(* CODESYS project GersSciPal_Project.project
   Company: io systems
   Title: GersSciPal_Project
   Description: application suivi de production
   Author: jl
   Version: 0.0.0.0

Project tree, tasks and I/O mapping:
  HMISCUxA5 : HMISCUxA5, Schneider Electric, order no. HMISCUxA5, version 3.5.3.59
      settings: OpcUa Enable = False
    application Application
      libraries: SysTimeRtc, 3.5.1.0 (System); ModbusTCP Slave, 3.5.3.50 (3S - Smart Software Solutions GmbH); 3S Storage, 3.5.3.0 (3S - Smart Software Solutions GmbH); BASIC, 3.3.4.0 (OSCAT)
      task MAST (cyclic, interval 20 ms, priority 15, watchdog 100 ms x 1) calls Prog_Main
      program Prog_Main [LD]
      Symbols
      999 - simulations/
        program random [LD]
        function block simulCounter [ST]
      200 - events & fifo/
        function block FB_fifoPushEvent [ST]
        program fifoManager [ST]
        function block eventManager [ST]
        function FC_fifoPush [ST]
      900 - utils/
        function CheckBounds [ST]
        function block TP_GSP [ST]
        function block Etat_Voyants [ST]
        function block counterWatch [ST]
        program CommunicationLife [ST]
      000 - data/
        global variables GVL
        data type _structModbusIn
        data type _structMessage
        data type alarmes
        data type _structVoyant
        data type _structModbusOut
        data type _structModbus
        data type _structIHMOFManager
        data type _structModbusMessage
      100 - time & com/
        program Modbus [LD]
        program timestamps [LD]
      300 - production/
        function block fabricationOrderManagement [ST]
    HMI Application
    Fonctions intégrées
      ES : ES, Schneider Electric, order no. IO, version 3.5.3.59
          input  iwES_Entr_e : WORD  // In
          output qwES_Sortie : WORD  // Out
      HSC : HSC, Schneider Electric, order no. HSC, version 3.5.3.59
      PTO_PWM : PTO_PWM, Schneider Electric, order no. PTO_PWM, version 3.5.3.59
    COM1
      SoMachine_Network_Manager : SoMachine-Network Manager, Schneider Electric, version 4.0.0.2
    Ethernet
      SoMachine_Network_Manager1 : SoMachine-Network Manager, Schneider Electric, version 4.0.0.2
    USB
      SoMachine_Network_Manager2 : SoMachine-Network Manager, Schneider Electric, version 4.0.0.2
    CAN
  Vijeo Designer Project Container Data
  Vijeo Designer Project Container
*)

// HMISCUxA5/Application/000 - data/_structModbusIn
TYPE _structModbusIn :
STRUCT
	ID: UDINT; // IDENTIFIANT DU MESSAGE AUTOMATE   0 à 3
    STATUT: INT; // ETAT A PRENDRE EN COMPTE         4 à 5
    lifeWD: INT; // MOT DE VIE  6 à 7
	rate: INT; // CADENCE THEORIQUE DE LA LIGNE
	reserve: INT;
END_STRUCT
END_TYPE

// HMISCUxA5/Application/000 - data/_structMessage
TYPE _structMessage :
STRUCT
	ihmOperations: STRING[8];
	ihmAlea: STRING[8];
	ihmLabels: STRING[32];

END_STRUCT
END_TYPE

// HMISCUxA5/Application/000 - data/alarmes
TYPE alarmes :
STRUCT
	attenteServeur: BOOL;
	attenteMariadb: BOOL;
	blocageMachine: BOOL;
	blocEvent: BOOL;
	blocOF: BOOL;
	nodeREDLife: BOOL;
END_STRUCT
END_TYPE

// HMISCUxA5/Application/000 - data/_structVoyant
TYPE _structVoyant :
STRUCT
	input: BOOL;
	change: BOOL;
	valeur: int;
END_STRUCT
END_TYPE

// HMISCUxA5/Application/000 - data/_structModbusOut
TYPE _structModbusOut :
STRUCT
	// VALEURS DES COMPTEURS
	CNT1: UDINT; // NOMBRE DE PIECES PRODUITES // de l'octet 8 à 11
	CNT2: UDINT; // NOMBRE DE PIECES PRODUITES MAIS PAS BONNES // de l'octet 12 à 15      
	
	// CONTENU DU MESSAGE
	MESSAGE: _structModbusMessage;
	
	// CADENCES ET SURVEILLANCES
	RUN: INT; // 2 octets - 74 à 75
	CRTHORODATAGE : UDINT; // 4 octets - 76 à 79
	CADENCE: UDINT;  // UNITE PAR HEURE --> CHRONO ENTRE DEUX PALETTE, TOUTES LES 2 MINUTES ON ENREGISTRE LA VALEUR DE CNT1 ; 4 octets - 80 à 83
	CADENCE_MOYENNE: UDINT; // UNITE PAR HEURE --> DIFFERENCE EN CNT1 ACTUEL - CNT1 D'IL Y A UNE HEURE ; 4 octets - 84 à 87 
	life: INT; // MOT DE VIE ; 2 octets - 88 à 89

END_STRUCT
END_TYPE

// HMISCUxA5/Application/000 - data/_structModbus
TYPE _structModbus :
STRUCT
	modbusIn: _structModbusIn;
	modbusOut: _structModbusOut;
END_STRUCT
END_TYPE

// HMISCUxA5/Application/000 - data/_structIHMOFManager
TYPE _structIHMOFManager :
	STRUCT
		startOF: BOOL; // commande démarrer OF
		stopOF: BOOL; // commande arrêter OF
		X0: BOOL; // attente lancement OF
		X1: BOOL; // lancement OF
		X2: BOOL; // OF en cours, attente arrêt OF
		X3: BOOL; // arrêt OF
		newOFEmpty: BOOL;
		seq: INT; // image du sequenceur
		newOF: STRING[12]; // nouvel OF à lancer
		cnt2: INT; // nombre de pièces défectueuses, saisi à l'arrêt de l'OF
	END_STRUCT
END_TYPE

// HMISCUxA5/Application/000 - data/_structModbusMessage
TYPE _structModbusMessage :
STRUCT
	ID: UDINT := 0; // 4 octets - 16 à 19
    STATUT: INT := 0; // 2 octets - 20 à 21
    OFNR: STRING[12] := '            '; // 13 octets - 22 à 33
    CODEM: STRING[8] := '        '; // 9 octets - 34 à 42
    OPERATION: STRING[8] := '        '; // 9 octets - 43 à 51
    ALEA: STRING[8] := '        '; // 9 octets - 52 à 60
    LIBELLE: STRING[32] := '                                '; // 17 octets - 52 à 67
	HORODATAGE: UDINT := 0; // 4 octets - 68 à 71 
	VALEUR: INT := 0; // 2 octets - 72 à 73
END_STRUCT
END_TYPE

// HMISCUxA5/Application/000 - data/GVL
VAR_GLOBAL
	Unixtime: UDINT; // Nombre de secondes depuis le 1er janvier 1970, lu sur l’horloge RTC de l’automate
	plcCycleTime: TIME;
	
	// table d'échange modbus avec Node-RED
	modbusInOut: _structModbus;
	startModbus: BOOL := TRUE;
	modbusError: BOOL := false;
	
	// données des messages et contenu de la FIFO
    fifoCount: INT := 0; // LONGUEUR REELLE DE LA PILE FIFO
	emptyMessage: _structModbusMessage; // CE MESSAGE DOIT TOUJOURS RESTER VIDE
	fifo: ARRAY[0..31] OF _structModbusMessage;
	
	// numéro d'OF de l'application
	OFNR: STRING[12] := '            ';
	
	// messages d'alarmes
	alm: alarmes;
	RPIOK: BOOL;
	DBOK: BOOL;
	NODEREDOK: BOOL;
	
	//Valeur Bouton IHM
	initFifoCount: BOOL;
	runAuto: BOOL;
	ihmButtons: ARRAY[0..15] OF BOOL;
	ihmOFManager: _structIHMOFManager;
	ihmOFRunning : BOOL;
	
	// gestion popup statut message
	closePopup: BOOL;
	
	// données gestion des voyants
	etatsVoyants: ARRAY[0..15] OF _structVoyant;
	
	// blocage machine
	AutorisationAuto AT %QX0.2 : BOOL;
	
END_VAR

VAR_GLOBAL CONSTANT
	fifoIndexMin: INT := 0;
    fifoIndexMax: INT := 31;
END_VAR

VAR_GLOBAL RETAIN PERSISTENT
	bypassAutoOut: BOOL;
	CNT1: UDINT;	// COMPTEUR DES PIECES CONFORMES
	CNT2: UDINT;	// COMPTEUR DES PIECES NON CONFORMES
	messageID: UDINT; // COMPTEUR DE MESSAGES
	CODEM: STRING[8];
	
	// PARAMETRES DE L'APPLICATION
	gvl_counterWatch_ptLife: TIME := T#20s;
	gvl_counterWatch_ptRate: TIME := T#2M;
	gvl_counterWatch_ptPercent: INT := 15;
	Param_minTime	: TIME := T#350MS;
	Param_maxTime	: TIME := T#750MS;
	Param_onOffTime	: TIME := T#2S;
	
	// RECETTE
	ihmMessages: ARRAY[0..31] OF _structMessage;
	
	// TITRES DES BOUTONS IHM
	buttons_FR: ARRAY[0..15] OF STRING[16];
	buttons_HU: ARRAY[0..15] OF STRING[16];
	buttons_EN: ARRAY[0..15] OF STRING[16];
	
END_VAR

// HMISCUxA5/Application/Prog_Main
PROGRAM Prog_Main
VAR
	
	em: eventManager;
	cw: counterWatch;
	fom: fabricationOrderManagement;
	
END_VAR

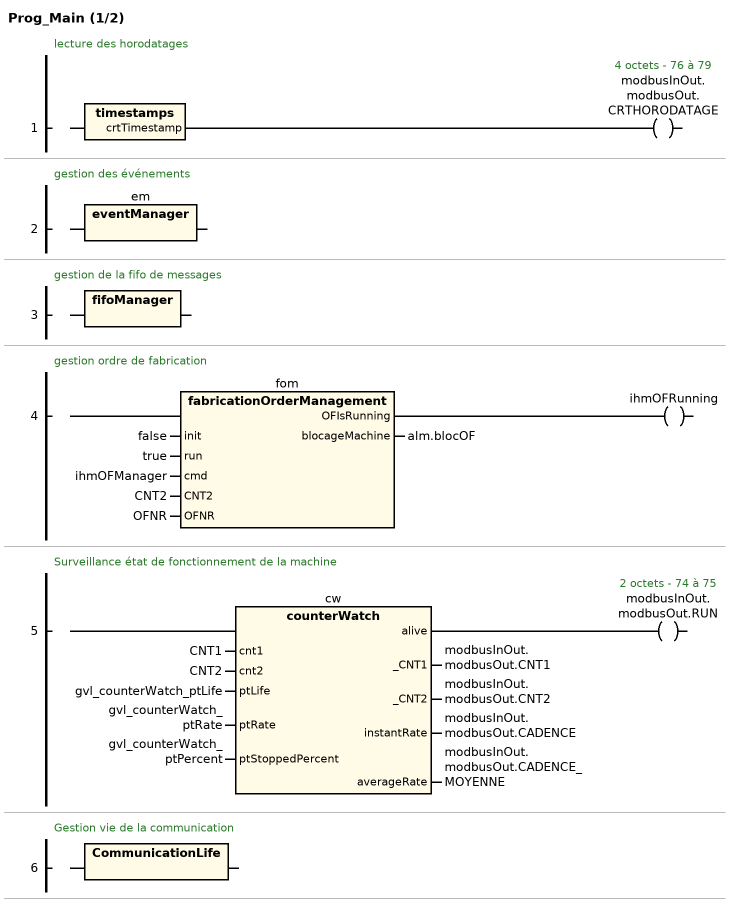
// NETWORK 1
// lecture des horodatages
//   modbusInOut.modbusOut.CRTHORODATAGE: 4 octets - 76 à 79
timestamps();
modbusInOut.modbusOut.CRTHORODATAGE := timestamps.crtTimestamp;

// NETWORK 2
// gestion des événements
em(); // eventManager

// NETWORK 3
// gestion de la fifo de messages
fifoManager();

// NETWORK 4
// gestion ordre de fabrication
//   CNT2: COMPTEUR DES PIECES NON CONFORMES
//   OFNR: numéro d'OF de l'application
fom(
    init := false,
    run := true,
    cmd := ihmOFManager,
    CNT2 := CNT2,
    OFNR := OFNR,
    blocageMachine => alm.blocOF); // fabricationOrderManagement
ihmOFRunning := fom.OFIsRunning;

// NETWORK 5
// Surveillance état de fonctionnement de la machine
//   CNT1: COMPTEUR DES PIECES CONFORMES
//   CNT2: COMPTEUR DES PIECES NON CONFORMES
//   gvl_counterWatch_ptLife: PARAMETRES DE L'APPLICATION
//   modbusInOut.modbusOut.CNT1: NOMBRE DE PIECES PRODUITES // de l'octet 8 à 11
//   modbusInOut.modbusOut.CNT2: NOMBRE DE PIECES PRODUITES MAIS PAS BONNES // de l'octet 12 à 15
//   modbusInOut.modbusOut.CADENCE: UNITE PAR HEURE --> CHRONO ENTRE DEUX PALETTE, TOUTES LES 2 MINUTES ON ENREGISTRE LA VALEUR DE CNT1 ; 4 octets - 80 à 83
//   modbusInOut.modbusOut.CADENCE_MOYENNE: UNITE PAR HEURE --> DIFFERENCE EN CNT1 ACTUEL - CNT1 D'IL Y A UNE HEURE ; 4 octets - 84 à 87
//   modbusInOut.modbusOut.RUN: 2 octets - 74 à 75
cw(
    cnt1 := CNT1,
    cnt2 := CNT2,
    ptLife := gvl_counterWatch_ptLife,
    ptRate := gvl_counterWatch_ptRate,
    ptStoppedPercent := gvl_counterWatch_ptPercent,
    _CNT1 => modbusInOut.modbusOut.CNT1,
    _CNT2 => modbusInOut.modbusOut.CNT2,
    instantRate => modbusInOut.modbusOut.CADENCE,
    averageRate => modbusInOut.modbusOut.CADENCE_MOYENNE); // counterWatch
modbusInOut.modbusOut.RUN := cw.alive;

// NETWORK 6
// Gestion vie de la communication
CommunicationLife();

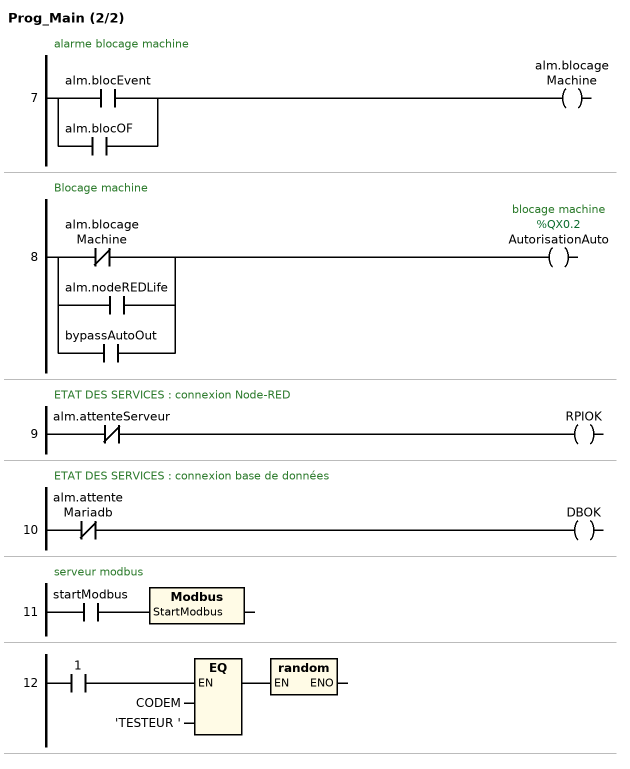
// NETWORK 7
// alarme blocage machine
alm.blocageMachine := alm.blocEvent OR alm.blocOF;

// NETWORK 8
// Blocage machine
//   AutorisationAuto: blocage machine | AT %QX0.2
AutorisationAuto := NOT alm.blocageMachine OR alm.nodeREDLife OR bypassAutoOut;

// NETWORK 9
// ETAT DES SERVICES : connexion Node-RED
RPIOK := NOT alm.attenteServeur;

// NETWORK 10
// ETAT DES SERVICES : connexion base de données
DBOK := NOT alm.attenteMariadb;

// NETWORK 11
// serveur modbus
Modbus(StartModbus := startModbus);

// NETWORK 12
IF 1 AND CODEM = 'TESTEUR ' THEN random(); END_IF

END_PROGRAM

// HMISCUxA5/Application/100 - time & com/timestamps
PROGRAM timestamps
VAR_OUTPUT
	crtTimestamp: UDINT;
END_VAR
VAR
	pResult :UDINT;
	tBool: BOOL;
	plcCyleTime: OSCAT_BASIC.CYCLE_TIME;
	ct_min: TIME;
	ct_max: TIME;
	systime: TIME;
	sysdays: INT;
	cycles:DWORD;
	tmpTime: DWORD;
END_VAR

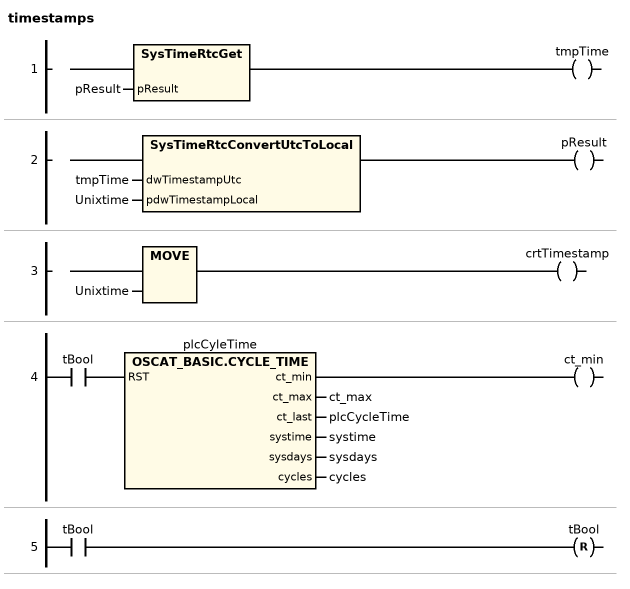
// NETWORK 1
tmpTime := SysTimeRtcGet(pResult := pResult);

// NETWORK 2
//   Unixtime: Nombre de secondes depuis le 1er janvier 1970, lu sur l’horloge RTC de l’automate
pResult := SysTimeRtcConvertUtcToLocal(dwTimestampUtc := tmpTime, pdwTimestampLocal := Unixtime);

// NETWORK 3
//   Unixtime: Nombre de secondes depuis le 1er janvier 1970, lu sur l’horloge RTC de l’automate
crtTimestamp := Unixtime;

// NETWORK 4
plcCyleTime(
    RST := tBool,
    ct_max => ct_max,
    ct_last => plcCycleTime,
    systime => systime,
    sysdays => sysdays,
    cycles => cycles); // OSCAT_BASIC.CYCLE_TIME
ct_min := plcCyleTime.ct_min;

// NETWORK 5
tBool R= tBool;

END_PROGRAM

// HMISCUxA5/Application/200 - events & fifo/eventManager
FUNCTION_BLOCK eventManager
VAR_INPUT
END_VAR
VAR_OUTPUT
END_VAR
VAR
	fifoPush: ARRAY[0..31] OF FB_fifoPushEvent;
	etatsVoyantsFB: ARRAY[0..15] OF Etat_Voyants;
	oldTmpBool: ARRAY[0..31] OF BOOL;
	tmpMessage: _structModbusMessage;
	tonResetButton11: Standard.TON;
	seqStop: INT := 0;
	msgIdStop: INT := 0;
END_VAR
VAR_TEMP
	tmpBool: BOOL;
	i: INT := 0;
	j: INT := 7;
END_VAR

tonResetButton11(in := ihmButtons[11], pt := T#500MS);
IF tonResetButton11.Q THEN
	ihmButtons[11] := FALSE;
END_IF

FOR i := 0 TO 31 BY +1 DO
	// SELECTION DE L'ENTREE AUTOMATE OU DU BOUTON IHM
	CASE i OF
		0: tmpBool:= %IX0.0;		
		1: tmpBool:= %IX0.1;		
		2: tmpBool:= %IX0.2;		
		3: tmpBool:= %IX0.3; 	
		4: tmpBool:= %IX0.4;		
		5: tmpBool:= %IX0.5;		
		6: tmpBool:= %IX0.6;		
		7: tmpBool:= %IX0.7;		
		8: tmpBool:= %IX1.0;
		9: tmpBool:= %IX1.1;
		10: tmpBool:= %IX1.2;
		11: tmpBool:= %IX1.3;
		12: tmpBool:= %IX1.4;
		13: tmpBool:= %IX1.5;
		14: tmpBool:= %IX1.6;
		15: tmpBool:= %IX1.7;
		16..31: tmpBool:= ihmButtons[i - 16];
	END_CASE
	
	// TRAITEMENT CAS PARTICULIER : OPERATION COMPTEUR
	IF ihmMessages[i].ihmOperations = 'COMPTEUR' THEN 
		
		// UNIQUEMENT ENTREE AUTOMATE
		IF i < 16 THEN
			// COMPTEUR DES PIECES CONFORMES
			IF ihmMessages[i].ihmAlea = 'CNT1    ' THEN
				IF tmpBool AND NOT oldTmpBool[i] THEN
					CNT1 := CNT1 + 1;
				END_IF;

			// COMPTEUR DES PIECES NON CONFORMES
			ELSIF ihmMessages[i].ihmAlea = 'CNT2    ' THEN
				IF tmpBool AND NOT oldTmpBool[i] THEN
					CNT2 := CNT2 + 1;
				END_IF;
			END_IF;
			
		END_IF;

	// TRAITEMENT CAS PARTICULIER : ENTREE AUTOMATE IMAGE D'UN VOYANT
	ELSIF ihmMessages[i].ihmOperations = 'VOYANT  ' THEN 
		
		// UNIQUEMENT ENTREE AUTOMATE
		IF i < 16 THEN
			// fonction de gestion de voyant
			etatsVoyantsFB[i](input := tmpBool, etatV := etatsVoyants[i]); 
		
			// DETECTION DERNIER CARACTERE DE LA CHAINE ALEA
			FOR j := 7 TO 0 BY -1 DO  
				IF ihmMessages[i].ihmAlea[j] <> 32 THEN
					EXIT;
				END_IF;
			END_FOR;
			// ECRITURE DE LA VALEUR DU VOYANT
			ihmMessages[i].ihmAlea[j] := BYTE#48 + INT_TO_BYTE(etatsVoyants[i].valeur); 
			
			// INSERTION DU MESSAGE DANS LA FIFO
			fifoPush[i](
				insert := etatsVoyants[i].change, 
				message:= ihmMessages[i]
			);
		END_IF;
		
	// TRAITEMENT CAS PARTICULIER : MESSAGES SYSTEME
	ELSIF ihmMessages[i].ihmOperations = 'RUN     ' THEN
		
		// MESSAGE 'RUNAUTO'
		IF ihmMessages[i].ihmAlea = 'RUNAUTO ' THEN
			tmpBool := modbusInOut.modbusOut.RUN > 0;
			fifoPush[i](
				insert := tmpBool,
				message:= ihmMessages[i]
			);
			
			// Blocage fonctionnement machine sur front descendant état de marche machine
			IF NOT tmpBool AND oldTmpBool[i] THEN
				seqStop := 1;
				// mémorisation horodatage arrêt machine
				tmpMessage.HORODATAGE := Unixtime;
				
			ELSIF tmpBool AND NOT oldTmpBool[i] AND seqStop = 1 THEN
				ihmButtons[11] := TRUE;
				
			END_IF; 
			
		END_IF;
		
	// CAS GENERAL : ENTREES AUTOMATE, NE DEBLOQUENT PAS LA MACHINE
	ELSIF i < 16 THEN
		// cas général
		fifoPush[i](
			insert := tmpBool,
			message:= ihmMessages[i]
		);
		
	// CAS GENERAL : BOUTONS IHM
	ELSE
		CASE seqStop OF
			0: // cas général
				fifoPush[i](
					insert := tmpBool,
					message:= ihmMessages[i]
				);
			
			1: // machine bloquée, attente sélection bouton ou redémarrage machine
				IF tmpBool AND NOT oldTmpBool[i] THEN
					msgIdStop := i;
					tmpMessage.OPERATION := ihmMessages[i].ihmOperations;
					tmpMessage.ALEA := ihmMessages[i].ihmAlea;
					tmpMessage.LIBELLE := ihmMessages[i].ihmLabels;
					// tmpMessage.horodatage a été saisi au front montant de alm.blocEvent, ligne 82
					tmpMessage.VALEUR := 1;
					FC_fifoPush(
						message := tmpMessage
					);
					seqStop := 2;
				END_IF
				
			2: // machine bloquée, attente remise à 0 du bouton IHM
				IF i = msgIdStop AND NOT tmpBool AND oldTmpBool[i] THEN
					tmpMessage.OPERATION := ihmMessages[i].ihmOperations;
					tmpMessage.ALEA := ihmMessages[i].ihmAlea;
					tmpMessage.LIBELLE := ihmMessages[i].ihmLabels;
					tmpMessage.horodatage := Unixtime;
					tmpMessage.VALEUR := 0;
					FC_fifoPush(
						message := tmpMessage
					);
					seqStop := 0;
				END_IF
				
			ELSE
				seqStop := 0;
			
		END_CASE
		
	END_IF;
	
	// MISE A JOUR DES ETATS PRECEDENTS
	oldTmpBool[i] := tmpBool;
	
END_FOR
alm.blocEvent := seqStop >= 1;

// REMPLACEMENT CARACTERE 0 PAR UN ESPACE DANS LE CODEM (VENANT DE LA RECETTE)
FOR i := 0 TO 7 BY +1 DO
	IF CODEM[ i ] = 0 THEN
		CODEM[ i ] := 32;
	END_IF
END_FOR;

END_FUNCTION_BLOCK

// HMISCUxA5/Application/200 - events & fifo/FC_fifoPush
FUNCTION FC_fifoPush : int
VAR_INPUT
	message: _structModbusMessage;
END_VAR

// NE DOIT ETRE APPELEE QUE SUR FRONT MONTANT OU DESCENDANT !!!

IF message.OPERATION = '        ' OR message.ALEA = '        ' OR message.LIBELLE = '                                ' THEN
	RETURN;
END_IF

// ENREGISTREMENT DU MESSAGE
fifo[ fifoCount ] := message;

// MISE A JOUR DES VALEURS PAR DEFAUT
fifo[ fifoCount ].ID := messageID;
fifo[ fifoCount ].STATUT := 2;
fifo[ fifoCount ].OFNR := OFNR;
fifo[ fifoCount ].CODEM := CODEM;

// MISE À JOUR DE LA LONGUEUR DE LA PILE
IF fifoCount < fifoIndexMax THEN
	fifoCount := fifoCount + 1;
END_IF;

// INCRÉMENT DU COMPTEUR DE MESSAGE
messageID := messageID + 1;
IF messageID > 32765 THEN
	messageID := 0;
END_IF;

FC_fifoPush := 0;

END_FUNCTION

// HMISCUxA5/Application/200 - events & fifo/FB_fifoPushEvent
FUNCTION_BLOCK FB_fifoPushEvent
VAR_INPUT
	insert: BOOL;
	message: _structMessage;
END_VAR
VAR
	memInsert: BOOL;
END_VAR
VAR_TEMP
	tmpMessage: _structModbusMessage;
END_VAR

// CONTROLE DU CONTENU DU MESSAGE
IF message.ihmOperations = '        ' OR message.ihmAlea = '        ' OR message.ihmLabels = '                                '
	OR CODEM = '        ' THEN
	RETURN;
END_IF

// INSERTION MESSAGE SUR CHANGEMENT D'ETAT DE L'ENTREE INSERT
IF insert AND NOT memInsert  OR NOT insert AND memInsert THEN
	// DÉFINITION DU MESSAGE
	tmpMessage.OPERATION := message.ihmOperations;
	tmpMessage.ALEA := message.ihmAlea;
	tmpMessage.LIBELLE := message.ihmLabels;
	tmpMessage.HORODATAGE := Unixtime;
	IF insert THEN
		tmpMessage.VALEUR := 1;
	ELSE
		tmpMessage.VALEUR := 0;
	END_IF;
	
	FC_fifoPush(
		message := tmpMessage
	);

END_IF;
memInsert := insert;

END_FUNCTION_BLOCK

// HMISCUxA5/Application/900 - utils/Etat_Voyants
FUNCTION_BLOCK Etat_Voyants
VAR_INPUT
	input: BOOL;
END_VAR
VAR_IN_OUT
	etatV: _structVoyant;
END_VAR
VAR
	old_input: BOOL;
	tmp: INT := 0;
	old_tmp: INT := 0;
	time_on: TIME;
	time_off: TIME;
	last_time_on: TIME;
	last_time_off: TIME;
	tonChange : Standard.TON;
	seq: INT;
	backup: INT;
END_VAR
VAR_TEMP
	minTime		: TIME;
	maxTime		: TIME;
	onOffTime	: TIME;
	cycleTime	: TIME;
	limitTime	: TIME;
END_VAR

minTime := Param_minTime;// T#250MS;
maxTime := Param_maxTime; // T#500MS;
onOffTime := Param_onOffTime; // T#2S;
cycleTime := onOffTime; // Param_cycleTime; // T#2S;
limitTime := T#30S;

etatV.input := input;

IF etatv.input AND NOT old_input THEN
	last_time_off := time_off;
	time_off := T#0S;
END_IF
IF NOT etatv.input AND old_input THEN
	last_time_on := time_on;
	time_on := T#0S;
END_IF

IF etatv.input THEN
	IF time_on < limitTime THEN
		time_on := time_on + plcCycleTime;
	END_IF;
ELSE
	IF time_off < limitTime THEN
		time_off := time_off + plcCycleTime;
	END_IF;
END_IF

IF time_on > onOffTime THEN
	tmp := 1;
	
ELSIF time_off > onOffTime THEN
	tmp := 0;
	
ELSIF last_time_on > minTime AND last_time_off > minTime THEN
	IF last_time_on > maxTime AND last_time_off > maxTime THEN
		tmp := 3;
	ELSE
		tmp := 2;
	END_IF;
END_IF; 

tonChange(in := etatV.valeur <> tmp, pt := cycleTime);
CASE seq OF
	0: 
		IF tonChange.Q THEN
			old_tmp := etatV.valeur;
			backup := tmp;
			seq := 1;
		END_IF
		
	1: 
		etatV.change := FALSE;
		seq := 2;
		
	2:
		etatV.valeur := backup;
		etatV.change := TRUE;
		seq := 0;
		
	ELSE
		seq := 0;
			 
END_CASE

old_input := etatv.input;

END_FUNCTION_BLOCK

// HMISCUxA5/Application/200 - events & fifo/fifoManager
PROGRAM fifoManager
VAR
	i: INT;
	TON_STEP2: Standard.TON;
	TON_STEP3: Standard.TON;
	TON_STEP4: Standard.TON;
	TON_STEP6: Standard.TON;
	TON_STEP80: Standard.TON;
	TON_STEP81: Standard.TON;
	cycleTime: TIME := T#500MS;
	timeoutNodeRED: TIME := T#5S;
	timeoutDB: TIME := T#5S;
	resumeTime: TIME := T#2S;
	errServerCnt: INT := 0;
	errMariadDBCnt: INT := 0;
	maxErr: INT := 5;
END_VAR

// RECHERCHE DE L’INDICE DU PREMIER CHAMP VIDE EN PARTANT DU BAS DE LA PILE
// EXECUTER CETTE FONCTION UNIQUEMENT APRES LA MISE EN RUN DE L'AUTOMATE OU A LA DEMANDE
// PAR UN BOUTON IHM SI FIFOCOUNT EST PERDU
IF initFifoCount THEN
	FOR i := fifoIndexMax TO fifoIndexMin BY -1 DO
    	IF fifo[ i ].STATUT > 0 THEN
        	fifoCount := i + 1;
    	END_IF;
	END_FOR;	
	initFifoCount := FALSE;
END_IF

// TEMPORISATION CONTROLE COMMUNICATION
TON_STEP2( IN := fifo[ fifoIndexMin ].STATUT = 2, PT := cycleTime);
TON_STEP3( IN := fifo[ fifoIndexMin ].STATUT = 3, PT := timeoutNodeRED);
TON_STEP4( IN := fifo[ fifoIndexMin ].STATUT = 4, PT := timeoutDB);
TON_STEP6( IN := fifo[ fifoIndexMin ].STATUT = 6, PT := cycleTime);
TON_STEP80( IN := fifo[ fifoIndexMin ].STATUT = 80, PT := resumeTime);
TON_STEP81( IN := fifo[ fifoIndexMin ].STATUT = 81, PT := resumeTime);

// GESTION ACTIVITE PREMIER MESSAGE DANS LA FIFO
CASE fifo[ fifoIndexMin ].STATUT OF
	0:	// STATUS 0 = PAS DE MESSAGE
		;
		
	1:	// STATUS 1 = MESSAGE EN COURS DE SAISIE 
		;
		
	2: 	// STATUS 2 = MESSAGE EN ATTENTE DE TRANSMISSION
		IF TON_STEP2.Q THEN
			// MISE À DISPOSITION DU PREMIER MESSAGE DE LA PILE POUR SRV-IOT
			fifo[ fifoIndexMin ].STATUT := 3;
		END_IF;
		
	3:	// STATUS 3 = ATTENTE PRISE EN COMPTE MESSAGE PAR NODE-RED
		// SRV-IOT A LU LE MESSAGE
		IF modbusInout.modbusIn.ID = fifo[ fifoIndexMin ].ID AND modbusInout.modbusIn.STATUT = 4 THEN
			errServerCnt := 0;
			fifo[ fifoIndexMin ].STATUT := 4;
			
		ELSIF TON_STEP3.Q THEN
			// TIME OUT : Node-RED n'a pas répondu assez rapidement : annulation et relance
			errServerCnt := errServerCnt + 1;
			fifo[fifoIndexMin].STATUT := 80;
			
		END_IF;
		
	4: // STATUS 4 = ATTENTE RETOUR ENREGISTREMENT DANS LA BASE DE DONNEES
		alm.attenteServeur := FALSE;
		// LE MESSAGE A ÉTÉ ENREGISTRÉ DANS LA BASE DE DONNÉES
		IF modbusInout.modbusIn.ID = fifo[ fifoIndexMin ].ID AND modbusInout.modbusIn.STATUT = 5 THEN
			errMariadDBCnt := 0;
			fifo[ fifoIndexMin ].STATUT := 5;
			
		ELSIF TON_STEP4.Q THEN
			// TIME OUT : Node-RED n'a pas répondu dans les temps : annulation et relance
			errMariadDBCnt := errMariadDBCnt + 1;
			fifo[ fifoIndexMin ].STATUT := 81;
			
		END_IF;
		
	5:	// STATUS 5 = ARCHIVAGE MESSAGE ET ON PASSE AU SUIVANT
		alm.attenteMariadb := FALSE;
		// DECALAGE DE LA FIFO DE MESSAGES, ECRASEMENT DU MESSAGE EN COURS DE TRAITEMENT...
		FOR i := fifoIndexMin TO fifoIndexMax - 1 BY 1 DO
			fifo[ i ] := fifo[ i + 1];
		END_FOR;
		fifo[ fifoIndexMax ] := emptyMessage;
		
		// MISE À JOUR DE LA LONGUEUR RÉELLE DE LA PILE
		IF fifoCount > fifoIndexMin THEN
			fifoCount := fifoCount - 1;
		END_IF;
		
		// fermeture popup statut message
		closePopup := not closePopup;

	80:	// STATUT 80 : TIME OUT PRISE EN COMPTE DU MESSAGE PAR NODE RED
		alm.attenteServeur := TRUE;
		IF TON_STEP80.Q THEN
			fifo[ fifoIndexMin ].STATUT := 2;
		ELSIF errServerCnt >= maxErr THEN
			errServerCnt := 0;
			fifo[ fifoIndexMin ].STATUT := 5;
		END_IF;
		
	81: // STATUT 81 : TIME OUT ENREGISTREMENT MESSAGE DANS LA BASE DE DONNEES
		alm.attenteMariadb := TRUE;
		IF TON_STEP81.Q THEN
			fifo[ fifoIndexMin ].STATUT := 2;
		ELSIF errMariadDBCnt >= maxErr THEN
			errMariadDBCnt := 0;
			fifo[ fifoIndexMin ].STATUT := 5;
		END_IF;
		
	ELSE
		fifo[ fifoIndexMin ].STATUT := 0;
		
END_CASE;

// transmission message en modbus
modbusInOut.modbusOut.MESSAGE.STATUT := fifo[ fifoIndexMin ].STATUT;
IF fifo[ fifoIndexMin ].STATUT <= 0 THEN
	modbusInOut.modbusOut.MESSAGE.CODEM := CODEM;
	modbusInOut.modbusOut.MESSAGE.OFNR := OFNR;
	modbusInOut.modbusOut.MESSAGE.HORODATAGE := Unixtime;
ELSE
	modbusInOut.modbusOut.MESSAGE.ID :=  fifo[ fifoIndexMin ].ID;
	modbusInOut.modbusOut.MESSAGE.CODEM :=  fifo[ fifoIndexMin ].CODEM;
	modbusInOut.modbusOut.MESSAGE.OFNR :=  fifo[ fifoIndexMin ].OFNR;
	modbusInOut.modbusOut.MESSAGE.HORODATAGE :=  fifo[ fifoIndexMin ].HORODATAGE;
	modbusInOut.modbusOut.MESSAGE.OPERATION :=  fifo[ fifoIndexMin ].OPERATION;
	modbusInOut.modbusOut.MESSAGE.ALEA :=  fifo[ fifoIndexMin ].ALEA;
	modbusInOut.modbusOut.MESSAGE.LIBELLE :=  fifo[ fifoIndexMin ].LIBELLE;
	modbusInOut.modbusOut.MESSAGE.VALEUR :=  fifo[ fifoIndexMin ].VALEUR;
END_IF;

END_PROGRAM

// HMISCUxA5/Application/100 - time & com/Modbus
PROGRAM Modbus
VAR_IN_OUT
	StartModbus: BOOL;
END_VAR
VAR
	reset: BOOL;
	xBusy: BOOL;
	modbusInADR: POINTER TO WORD := ADR(modbusInOut);
	modbusRegistersADR: POINTER TO WORD:= ADR(modbusInOut.modbusIn.ID);
	ByClientConnection: BYTE;
	uiInputDataSize: UINT := 8; // A ADAPTER
	uiOutputDataSize: UINT := 108; // A ADAPTER
	TON_Start: TON;
	TON_Start_ET: TIME;
	ModbusServer_1 : ModbusServer;

END_VAR

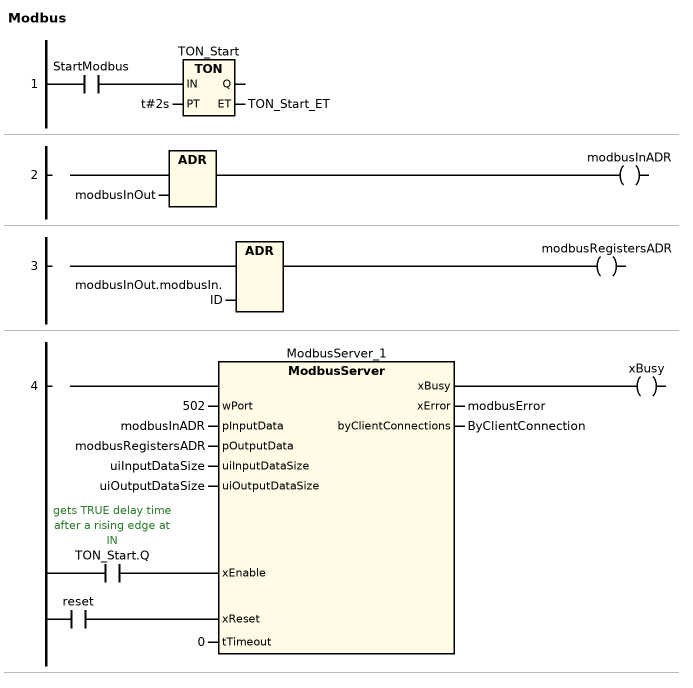
// NETWORK 1
TON_Start(IN := StartModbus, PT := t#2s, ET => TON_Start_ET); // TON

// NETWORK 2
//   modbusInOut: table d'échange modbus avec Node-RED
modbusInADR := ADR(modbusInOut);

// NETWORK 3
//   modbusInOut.modbusIn.ID: IDENTIFIANT DU MESSAGE AUTOMATE 0 à 3
modbusRegistersADR := ADR(modbusInOut.modbusIn.ID);

// NETWORK 4
//   uiInputDataSize: A ADAPTER
//   uiOutputDataSize: A ADAPTER
//   TON_Start.Q: gets TRUE delay time after a rising edge at IN
ModbusServer_1(
    wPort := 502,
    pInputData := modbusInADR,
    pOutputData := modbusRegistersADR,
    uiInputDataSize := uiInputDataSize,
    uiOutputDataSize := uiOutputDataSize,
    xEnable := TON_Start.Q,
    xReset := reset,
    tTimeout := 0,
    xError => modbusError,
    byClientConnections => ByClientConnection); // ModbusServer
xBusy := ModbusServer_1.xBusy;

END_PROGRAM

// HMISCUxA5/Application/300 - production/fabricationOrderManagement
FUNCTION_BLOCK fabricationOrderManagement
VAR_INPUT
	init: BOOL;
	run: BOOL;
END_VAR
VAR_OUTPUT
	OFIsRunning: BOOL;
	blocageMachine: BOOL;
END_VAR
VAR_IN_OUT
	cmd: _structIHMOFManager;
	CNT2: UDINT;
	OFNR: STRING[12];
END_VAR
VAR
	seq: INT;
END_VAR

// initialisations
OFIsRunning := FALSE;
blocageMachine := TRUE;

IF init THEN
	seq := 0;
	RETURN;
END_IF

// désactivation des transitions
IF NOT run THEN
	JMP end;
END_IF

// sequence
CASE seq OF
	0: // attente lancement OF
		IF cmd.newOF <> '            ' AND cmd.startOF THEN
			seq := 10;
		
		// si OF enregistré au démarrage, on l'arrête
		ELSIF OFNR <> '            ' THEN
			seq := 30;
			
		END_IF;
		
	10: // enregistrement du nouvel OF
		OFNR := cmd.newOF;
		cmd.startOF := FALSE;
		cmd.stopOF := FALSE;
		cmd.newOF := '            ';
		cmd.cnt2 := 0;
		seq := 20;
		
	20: // OF en cours
		OFIsRunning := TRUE;
		blocageMachine := FALSE;
		IF cmd.stopOF THEN
			seq := 30;
		END_IF;
		
	30: // arrêt OF en cours
		OFNR := '            ';
		cmd.startOF := FALSE;
		cmd.stopOF := FALSE;
		cmd.newOF := '            ';
		CNT2 := CNT2 + INT_TO_UDINT(cmd.cnt2);
		cmd.cnt2 := 0;
		seq := 0;
		
	ELSE
		seq := 0;
END_CASE

// mise à jour des recopies
end:
cmd.seq := seq / 10;
cmd.X0 := seq = 0;
cmd.X1 := seq = 10;
cmd.X2 := seq = 20;
cmd.X3 := seq = 30;
cmd.newOFEmpty := cmd.newOF = '            ';

END_FUNCTION_BLOCK

// HMISCUxA5/Application/900 - utils/counterWatch
FUNCTION_BLOCK counterWatch
VAR_INPUT
	cnt1: UDINT;
	cnt2: UDINT;
	ptLife: TIME;
	ptRate: TIME;
	ptStoppedPercent: INT;
END_VAR
VAR_OUTPUT
	alive: INT;
	_CNT1: UDINT;
	_CNT2: UDINT;
	instantRate: UDINT;
	averageRate: UDINT;
END_VAR
VAR
	TP_Life: TP_GSP;
	tonRate: TON;
	_ptLife: TIME;
	_ptRate: TIME;
	seq : INT;
	i : INT;
	tmpIndex: INT;
	oldCnt: UDINT;
	counts: ARRAY[0..59] OF UDINT;
	tmpReal: REAL;
END_VAR

// recopie des compteurs en sortie
_cnt1 := cnt1;
_cnt2 := cnt2;

// calcul du temps entre deux unités de cadences
_ptLife := ptLife;
IF modbusInOut.modbusIn.rate > 0 AND ptStoppedPercent > 0 AND  ptStoppedPercent < 100 THEN
	tmpReal := 3600.0 / (INT_TO_REAL(modbusInOut.modbusIn.rate) * (INT_TO_REAL(ptStoppedPercent) / 100.0)) * 1000.0; // Temps entre deux unités en millisecondes, temps mini = ptStoppedPercent de la cadence totale
	IF tmpReal > 0 THEN
		_ptLife := REAL_TO_TIME(tmpReal);
	END_IF
END_IF

// contrôle de la vie du compteur
TP_Life(in := cnt1 <> oldCnt, pt := _ptLife);
IF TP_Life.Q THEN
	alive := 1;
ELSE
	alive := 0;
END_IF
oldCnt := cnt1;

// init tableau en cas de remise à 0 du compteur
IF cnt1 < counts[0] THEN
	FOR i := 0 TO 29 BY 1 DO
		counts[i] := 0;
	END_FOR
END_IF

IF ptRate <= T#0S THEN
	return;
END_IF
_ptRate := ptRate;
IF _ptRate < T#1M THEN
	_ptRate := T#1M;
END_IF
IF _ptRate > T#1H THEN
	_ptRate := T#1H;
END_IF

// temps entre deux mesures de la cadence
tonRate(in := seq = 0, pt := _ptRate);

// séquence mesures de la cadence
CASE seq OF
	0:	// ATTENTE TEMPO CADENCE
		IF tonRate.Q THEN
			seq := 10;
		END_IF
		
	10: // INTEGRATION DE LA DERNIERE VALEUR DU COMPTEUR
		FOR i := 59 TO 1 BY -1 DO
			counts[i] := counts[i - 1];
		END_FOR
		counts[0] := cnt1;
		
		// CALCUL CADENCE INSTANTANEE
		// interdiction division par 0 et valeur négative
		IF _ptRate > T#0S AND counts[0] >= counts[1] THEN
			instantRate := (counts[0] - counts[1]) * TIME_TO_UDINT(T#1H) / TIME_TO_UDINT(_ptRate);
		ELSE
			instantRate := 0;
		END_IF
		
		// CALCUL DE LA CADENCE A L'HEURE
		// interdiction division par 0
		IF _ptRate > T#0S THEN
			tmpIndex := UDINT_TO_INT(TIME_TO_UDINT(T#1H) / TIME_TO_UDINT(_ptRate)) - 1;
			
			// tmpIndex doit être dans les limites du tableau
			IF tmpIndex > 0 AND tmpIndex <= 59 THEN
				
				// interdiction valeur négative
				IF counts[0] >= counts[tmpindex] THEN
					averageRate := (counts[0] - counts[tmpIndex]);
				ELSE
					averageRate := 0;
				END_IF
			ELSE
				averageRate := 0;
			END_IF;
		ELSE
			averageRate := 0;
		END_IF
		seq := 0;
		
	ELSE
		seq := 0;
END_CASE

END_FUNCTION_BLOCK

// HMISCUxA5/Application/900 - utils/TP_GSP
FUNCTION_BLOCK TP_GSP
VAR_INPUT
	IN: BOOL;
	PT: TIME;
END_VAR
VAR_OUTPUT
	Q: BOOL;
	ET: TIME;
END_VAR
VAR
	aux_in: BOOL;
	seq: INT;
	lastStart: TIME;
END_VAR

IF in AND NOT aux_in THEN
	lastStart := UDINT_TO_TIME(unixtime) * 1000;
	et := T#0s;
END_IF 
aux_in := in;

Q := FALSE;
CASE seq OF
	0:
		IF in THEN
			seq := 1;
		END_IF
		
	1:
		q := TRUE; 
		IF ET < PT THEN
			ET := UDINT_TO_TIME(unixtime) * 1000 - laststart;
		ELSE
			seq := 2;
		END_IF
		
	2:
		IF NOT in THEN
			seq := 0;
		END_IF
		
END_CASE

END_FUNCTION_BLOCK

// HMISCUxA5/Application/900 - utils/CommunicationLife
PROGRAM CommunicationLife
VAR
	oldReceivedLife: INT;
	seq: INT := 0;
	filterTime: TIME;
	TONLife: Standard.TON;
	TOFLife: Standard.TOF;
	ton_1: TON;
	ton_2: TON;
END_VAR

// création de la vie
IF modbusInOut.modbusOut.life < 999 THEN
	modbusInOut.modbusOut.life := modbusInOut.modbusOut.life + 1;
ELSE
	modbusInOut.modbusOut.life := 0;
END_IF

// surveillance vie Node-RED
filterTime := T#2S;
TONLife(in := modbusInOut.modbusIn.lifeWD = oldReceivedLife, pt := filterTime);
TOFLife(in := TONLife.Q, pt := filterTime);
oldReceivedLife := modbusInOut.modbusIn.lifeWD;

alm.nodeREDLife := FALSE; // TOFLife.Q;
NODEREDOK := NOT alm.nodeREDLife;

IF NODEREDOK THEN
	seq := 0;
	StartModbus := not modbusError;
	RETURN;
END_IF

ton_1(in := seq = 0 AND alm.nodeREDLife, pt := T#60S);
ton_2(in := seq = 1, pt := T#5S);

CASE seq OF
	0: // tempo avant désactivation modbus
		IF ton_1.Q THEN
			seq := 1;
		END_IF;
		
	1: // temps avant réactivation modbus
		IF ton_2.Q THEN
			seq := 0;
		END_IF;
		
	ELSE
		seq := 0;
END_CASE
StartModbus := seq = 0;

END_PROGRAM

// HMISCUxA5/Application/999 - simulations/random
PROGRAM random
VAR
	tonCadence: Standard.TON;
	cycleCadence: TIME := T#1M;
	
	localRUN: BOOL;
	minutes: INT; 
	tmpDINT: DINT;
	simul_01: simulCounter;
	
END_VAR
VAR // added by the converter: edge detectors and wires of the graphical bodies
    _w1, _w2 : BOOL;
END_VAR

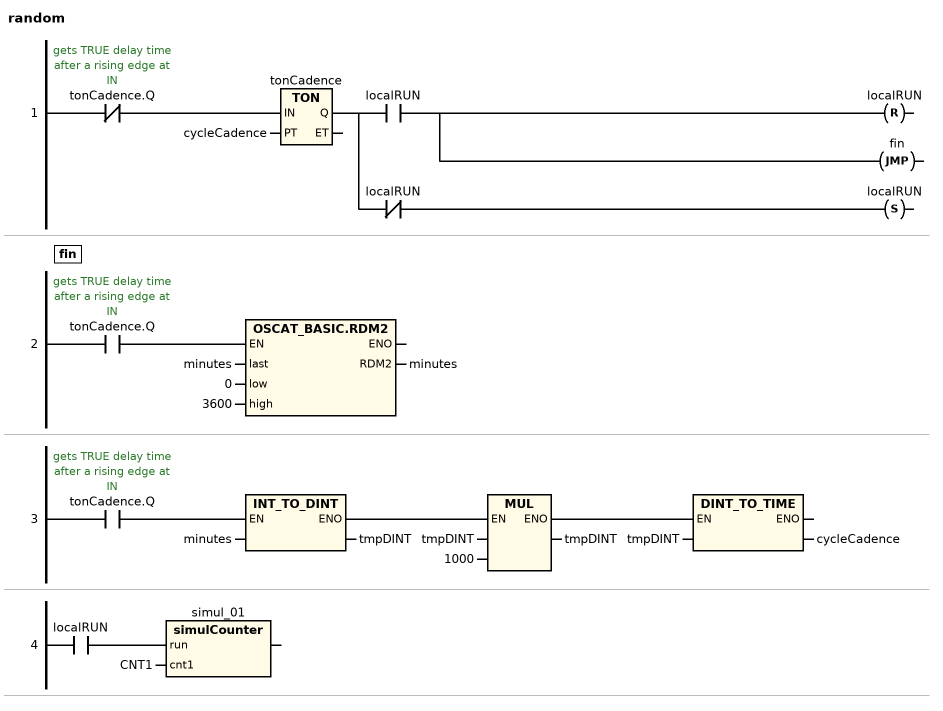
// NETWORK 1
//   tonCadence.Q: gets TRUE delay time after a rising edge at IN
tonCadence(IN := NOT tonCadence.Q, PT := cycleCadence); // TON
_w1 := tonCadence.Q AND localRUN;
localRUN R= _w1;
IF _w1 THEN JMP fin; END_IF
localRUN S= tonCadence.Q AND NOT localRUN;

// NETWORK 2
//   tonCadence.Q: gets TRUE delay time after a rising edge at IN
fin:
IF tonCadence.Q THEN minutes := OSCAT_BASIC.RDM2(last := minutes, low := 0, high := 3600); END_IF

// NETWORK 3
//   tonCadence.Q: gets TRUE delay time after a rising edge at IN
_w2 := tonCadence.Q;
IF _w2 THEN tmpDINT := INT_TO_DINT(minutes); END_IF
IF _w2 THEN tmpDINT := tmpDINT * 1000; END_IF
IF _w2 THEN cycleCadence := DINT_TO_TIME(tmpDINT); END_IF

// NETWORK 4
//   CNT1: COMPTEUR DES PIECES CONFORMES
simul_01(run := localRUN, cnt1 := CNT1); // simulCounter

END_PROGRAM

// HMISCUxA5/Application/999 - simulations/simulCounter
FUNCTION_BLOCK simulCounter
VAR_INPUT
	run: BOOL;
END_VAR
VAR_IN_OUT
	cnt1: UDINT;
END_VAR
VAR_OUTPUT
END_VAR
VAR
	aux_run: BOOL;
	cadence: UDINT;
	lastStart: UDINT;
	crtTime: UDINT;
	crtCntRun: UDINT;
END_VAR

cadence := 1000; // unité par heure

IF run AND NOT aux_run THEN
	lastStart := Unixtime;
END_IF

IF run THEN
	crtTime := Unixtime - lastStart;
	crtCntRun := cadence * crtTime / 3600;
	IF crtCntRun > 0 THEN
		cnt1 := cnt1 + crtCntRun;
		crtCntRun := 0;
		lastStart := Unixtime;
	END_IF
END_IF

IF NOT run AND aux_run THEN
	cnt1 := cnt1 + crtCntRun;
	crtCntRun := 0;
END_IF

aux_run := run;

END_FUNCTION_BLOCK

// HMISCUxA5/Application/900 - utils/CheckBounds
// Code généré automatiquement : NE PAS MODIFIER
FUNCTION CheckBounds : DINT
VAR_INPUT
	index, lower, upper: DINT;
END_VAR

// Code généré automatiquement : Il s’agit d’une proposition d’implémentation.
IF  index < lower THEN
	CheckBounds := lower;
ELSIF  index > upper THEN
	CheckBounds := upper;
ELSE  
	CheckBounds := index;
END_IF

END_FUNCTION
